// TwinCAT 3 PLC project PLC1
// ProgramVersion: 3.1.4020.4
// libraries:
//   Tc2_MC2, * (Beckhoff Automation GmbH)
//   Tc2_Standard, * (Beckhoff Automation GmbH)
//   Tc2_System, * (Beckhoff Automation GmbH)
//   Tc2_Utilities, * (Beckhoff Automation GmbH)
//   Tc3_MC2_AdvancedHoming, * (Beckhoff Automation GmbH)
//   Tc3_Module, * (Beckhoff Automation GmbH)
//   Festo TcMC Library for TwinCAT 3,3.1.1,Festo AG & Co. KG
// project tree:
//   DataType/ MoveState_t.TcDUT
//   / PlcTask.TcTTO (not stored)
//   POUs/ AxisCtrl.TcPOU, MAIN.TcPOU
// real-time tasks:
//   TASK PlcTask: cycle T#10ms, priority 20, ADS port 350
// motion (NC):
//   TASK NC-Task 1 SAF: cycle T#2ms, priority 4, ADS port 501
//   TASK NC-Task 1 SVB: cycle T#10ms, priority 8, ADS port 511
//   AXIS Axis 1 (id 1)
//     Dynamic: AccelerationMaximum=20000, DecelerationMaximum=20000, Acceleration=10000, Deceleration=10000, Jerk=200000
//     Velo: FastManual=300, Maximum=1000
//     OtherSettings: AllowMotionCmdToSlave=true
//     encoder EncType=19
//       EncPara: ScaleFactorNumerator=90, ScaleFactorDenominator=65536, MaxCount=#xffffffff
//         Inc: RefSearchInverse=true, RefMode=5
//     drive DrvType=16
//       DrvPara: MaxCount=#xffffffff, DriveControlDWord=#x00000100
//         Analog: VeloReferenz=1100
//         TimeComp: TaskDelayCycles=1
//     controller CtrType=1
//       CtrPara: PriorControlFactor=1
//         Observer: BandWidth=20
//   AXIS Axis 2 (id 2)
//     Dynamic: AccelerationMaximum=20000, DecelerationMaximum=20000, Acceleration=10000, Deceleration=10000, Jerk=200000
//     Velo: Maximum=1000
//     OtherSettings: AllowMotionCmdToSlave=true
//     encoder EncType=19
//       EncPara: ScaleFactorNumerator=90, ScaleFactorDenominator=65536, MaxCount=#xffffffff
//         Inc: RefSearchInverse=true
//     drive DrvType=16
//       DrvPara: MaxCount=#xffffffff, DriveControlDWord=#x00000100
//         Analog: VeloReferenz=1100
//         TimeComp: TaskDelayCycles=1
//     controller CtrType=1
//       CtrPara: PriorControlFactor=1
//         Observer: BandWidth=20
//   AXIS Axis 3 (id 3)
//     Dynamic: AccelerationMaximum=20000, DecelerationMaximum=20000, Acceleration=10000, Deceleration=10000, Jerk=200000
//     Velo: Maximum=1000
//     OtherSettings: AllowMotionCmdToSlave=true
//     encoder EncType=1
//       EncPara: ScaleFactorNumerator=90, ScaleFactorDenominator=65536
//         Inc: RefSearchInverse=true
//     drive DrvType=5
//       Analog: VeloReferenz=1100
//       TimeComp: TaskDelayCycles=1
//     controller CtrType=1
//       CtrPara: PriorControlFactor=1
//         Observer: BandWidth=20
//   AXIS Axis 4 (id 4)
//     Dynamic: AccelerationMaximum=20000, DecelerationMaximum=20000, Acceleration=10000, Deceleration=10000, Jerk=200000
//     Velo: Maximum=1000
//     OtherSettings: AllowMotionCmdToSlave=true
//     encoder EncType=1
//       EncPara: ScaleFactorNumerator=90, ScaleFactorDenominator=65536
//         Inc: RefSearchInverse=true
//     drive DrvType=5
//       Analog: VeloReferenz=1100
//       TimeComp: TaskDelayCycles=1
//     controller CtrType=1
//       CtrPara: PriorControlFactor=1
//         Observer: BandWidth=20
//   AXIS Axis 5 (id 5)
//     Dynamic: AccelerationMaximum=20000, DecelerationMaximum=20000, Acceleration=10000, Deceleration=10000, Jerk=200000
//     Velo: Maximum=1000
//     OtherSettings: AllowMotionCmdToSlave=true
//     encoder EncType=1
//       EncPara: ScaleFactorNumerator=90, ScaleFactorDenominator=65536
//         Inc: RefSearchInverse=true
//     drive DrvType=5
//       Analog: VeloReferenz=1100
//       TimeComp: TaskDelayCycles=1
//     controller CtrType=1
//       CtrPara: PriorControlFactor=1
//         Observer: BandWidth=20
//   AXIS Axis 6 (id 6)
//     Dynamic: AccelerationMaximum=20000, DecelerationMaximum=20000, Acceleration=10000, Deceleration=10000, Jerk=200000
//     Velo: Maximum=1000
//     OtherSettings: AllowMotionCmdToSlave=true
//     encoder EncType=1
//       EncPara: ScaleFactorNumerator=90, ScaleFactorDenominator=65536
//         Inc: RefSearchInverse=true
//     drive DrvType=5
//       Analog: VeloReferenz=1100
//       TimeComp: TaskDelayCycles=1
//     controller CtrType=1
//       CtrPara: PriorControlFactor=1
//         Observer: BandWidth=20
//   AXIS Axis 7 (id 7)
//     Dynamic: AccelerationMaximum=20000, DecelerationMaximum=20000, Acceleration=10000, Deceleration=10000, Jerk=200000
//     Velo: Maximum=1000
//     OtherSettings: AllowMotionCmdToSlave=true
//     encoder EncType=1
//       EncPara: ScaleFactorNumerator=90, ScaleFactorDenominator=65536
//         Inc: RefSearchInverse=true
//     drive DrvType=5
//       Analog: VeloReferenz=1100
//       TimeComp: TaskDelayCycles=1
//     controller CtrType=1
//       CtrPara: PriorControlFactor=1
//         Observer: BandWidth=20
//   AXIS Axis 8 (id 8)
//     Dynamic: AccelerationMaximum=20000, DecelerationMaximum=20000, Acceleration=10000, Deceleration=10000, Jerk=200000
//     Velo: Maximum=1000
//     OtherSettings: AllowMotionCmdToSlave=true
//     encoder EncType=1
//       EncPara: ScaleFactorNumerator=90, ScaleFactorDenominator=65536
//         Inc: RefSearchInverse=true
//     drive DrvType=5
//       Analog: VeloReferenz=1100
//       TimeComp: TaskDelayCycles=1
//     controller CtrType=1
//       CtrPara: PriorControlFactor=1
//         Observer: BandWidth=20
//   AXIS Axis 9 (id 9)
//     Dynamic: AccelerationMaximum=20000, DecelerationMaximum=20000, Acceleration=10000, Deceleration=10000, Jerk=200000
//     Velo: Maximum=1000
//     OtherSettings: AllowMotionCmdToSlave=true
//     encoder EncType=1
//       EncPara: ScaleFactorNumerator=90, ScaleFactorDenominator=65536
//         Inc: RefSearchInverse=true
//     drive DrvType=5
//       Analog: VeloReferenz=1100
//       TimeComp: TaskDelayCycles=1
//     controller CtrType=1
//       CtrPara: PriorControlFactor=1
//         Observer: BandWidth=20
//   AXIS Axis 10 (id 10)
//     Dynamic: AccelerationMaximum=20000, DecelerationMaximum=20000, Acceleration=10000, Deceleration=10000, Jerk=200000
//     Velo: Maximum=1000
//     OtherSettings: AllowMotionCmdToSlave=true
//     encoder EncType=1
//       EncPara: ScaleFactorNumerator=90, ScaleFactorDenominator=65536
//         Inc: RefSearchInverse=true
//     drive DrvType=5
//       Analog: VeloReferenz=1100
//       TimeComp: TaskDelayCycles=1
//     controller CtrType=1
//       CtrPara: PriorControlFactor=1
//         Observer: BandWidth=20
// I/O:
//   DEVICE NIC, AmsNetId 192.168.2.43.2.1
//     Ctr1 [CMMP-AS V4p0 CiA402]
//     Ctr2 [CMMP-AS V4p0 CiA402]
// variable links:
//   NC-Task 1 SAF/Axes/Axis 1 <-> NIC/Ctr1
//     Drive/Inputs/In/nDataIn1 <-> Inputs_1/Following_Error_Actual_Value
//     Drive/Inputs/In/nDcOutputTime <-> InfoData/DcOutputShift
//     Drive/Inputs/In/nState1 <-> Inputs/Statusword
//     Drive/Inputs/In/nState2 <-> Inputs/Statusword @bit 8
//     Drive/Inputs/In/nState4 @bit 1 <-> WcState/InputToggle
//     Drive/Inputs/In/nState4 <-> WcState/WcState
//     Drive/Outputs/Out/nCtrl1 <-> Outputs/Controlword
//     Drive/Outputs/Out/nCtrl2 <-> Outputs/Controlword @bit 8
//     Drive/Outputs/Out/nDataOut1 <-> Outputs/IP_Data_Record
//     Enc/Inputs/In/nDataIn1 <-> Inputs/Position_Actual_Value
//     Enc/Inputs/In/nDcInputTime <-> InfoData/DcInputShift
//     Enc/Inputs/In/nState4 @bit 1 <-> WcState/InputToggle
//     Enc/Inputs/In/nState4 <-> WcState/WcState
//   NC-Task 1 SAF/Axes/Axis 2 <-> NIC/Ctr2
//     Drive/Inputs/In/nDataIn1 <-> Inputs_1/Following_Error_Actual_Value
//     Drive/Inputs/In/nDcOutputTime <-> InfoData/DcOutputShift
//     Drive/Inputs/In/nState1 <-> Inputs/Statusword
//     Drive/Inputs/In/nState2 <-> Inputs/Statusword @bit 8
//     Drive/Inputs/In/nState4 @bit 1 <-> WcState/InputToggle
//     Drive/Inputs/In/nState4 <-> WcState/WcState
//     Drive/Outputs/Out/nCtrl1 <-> Outputs/Controlword
//     Drive/Outputs/Out/nCtrl2 <-> Outputs/Controlword @bit 8
//     Drive/Outputs/Out/nDataOut1 <-> Outputs/IP_Data_Record
//     Enc/Inputs/In/nDataIn1 <-> Inputs/Position_Actual_Value
//     Enc/Inputs/In/nDcInputTime <-> InfoData/DcInputShift
//     Enc/Inputs/In/nState4 @bit 1 <-> WcState/InputToggle
//     Enc/Inputs/In/nState4 <-> WcState/WcState
//   PLC1/PLC1 Instance <-> NIC/Ctr1
//     PlcTask Inputs/MAIN.axisCtrls[1].amsAddr <-> InfoData/AdsAddr
//     PlcTask Inputs/MAIN.axisCtrls[1].dig_in <-> Input3/swn
//   PLC1/PLC1 Instance <-> NIC/Ctr2
//     PlcTask Inputs/MAIN.axisCtrls[2].amsAddr <-> InfoData/AdsAddr
//   PLC1/PLC1 Instance <-> NC-Task 1 SAF/Axes/Axis 1
//     PlcTask Inputs/MAIN.axisCtrls[1].axis.NcToPlc <-> Outputs/ToPlc
//     PlcTask Outputs/MAIN.axisCtrls[1].axis.PlcToNc <-> Inputs/FromPlc
//   PLC1/PLC1 Instance <-> NC-Task 1 SAF/Axes/Axis 10
//     PlcTask Inputs/MAIN.axisCtrls[10].axis.NcToPlc <-> Outputs/ToPlc
//     PlcTask Outputs/MAIN.axisCtrls[10].axis.PlcToNc <-> Inputs/FromPlc
//   PLC1/PLC1 Instance <-> NC-Task 1 SAF/Axes/Axis 2
//     PlcTask Inputs/MAIN.axisCtrls[2].axis.NcToPlc <-> Outputs/ToPlc
//     PlcTask Outputs/MAIN.axisCtrls[2].axis.PlcToNc <-> Inputs/FromPlc
//   PLC1/PLC1 Instance <-> NC-Task 1 SAF/Axes/Axis 3
//     PlcTask Inputs/MAIN.axisCtrls[3].axis.NcToPlc <-> Outputs/ToPlc
//     PlcTask Outputs/MAIN.axisCtrls[3].axis.PlcToNc <-> Inputs/FromPlc
//   PLC1/PLC1 Instance <-> NC-Task 1 SAF/Axes/Axis 4
//     PlcTask Inputs/MAIN.axisCtrls[4].axis.NcToPlc <-> Outputs/ToPlc
//     PlcTask Outputs/MAIN.axisCtrls[4].axis.PlcToNc <-> Inputs/FromPlc
//   PLC1/PLC1 Instance <-> NC-Task 1 SAF/Axes/Axis 5
//     PlcTask Inputs/MAIN.axisCtrls[5].axis.NcToPlc <-> Outputs/ToPlc
//     PlcTask Outputs/MAIN.axisCtrls[5].axis.PlcToNc <-> Inputs/FromPlc
//   PLC1/PLC1 Instance <-> NC-Task 1 SAF/Axes/Axis 6
//     PlcTask Inputs/MAIN.axisCtrls[6].axis.NcToPlc <-> Outputs/ToPlc
//     PlcTask Outputs/MAIN.axisCtrls[6].axis.PlcToNc <-> Inputs/FromPlc
//   PLC1/PLC1 Instance <-> NC-Task 1 SAF/Axes/Axis 7
//     PlcTask Inputs/MAIN.axisCtrls[7].axis.NcToPlc <-> Outputs/ToPlc
//     PlcTask Outputs/MAIN.axisCtrls[7].axis.PlcToNc <-> Inputs/FromPlc
//   PLC1/PLC1 Instance <-> NC-Task 1 SAF/Axes/Axis 8
//     PlcTask Inputs/MAIN.axisCtrls[8].axis.NcToPlc <-> Outputs/ToPlc
//     PlcTask Outputs/MAIN.axisCtrls[8].axis.PlcToNc <-> Inputs/FromPlc
//   PLC1/PLC1 Instance <-> NC-Task 1 SAF/Axes/Axis 9
//     PlcTask Inputs/MAIN.axisCtrls[9].axis.NcToPlc <-> Outputs/ToPlc
//     PlcTask Outputs/MAIN.axisCtrls[9].axis.PlcToNc <-> Inputs/FromPlc

// ---- DataType/MoveState_t.TcDUT
TYPE MoveState_t :
(
	 MOVESTATE_RESET,
	 MOVESTATE_INIT,
	 MOVESTATE_ENABLE,
	 MOVESTATE_HOMING,
	 MOVESTATE_MOVING,
	 MOVESTATE_ERROR	
);
END_TYPE

// ---- POUs/AxisCtrl.TcPOU
FUNCTION_BLOCK AxisCtrl
VAR_INPUT
END_VAR
VAR_OUTPUT
END_VAR
VAR
	axis : AXIS_REF;
	state : MoveState_t;
	
	moveAbs: MC_MoveAbsolute;
	moveAbsOut: ST_McOutputs;

	moveAbs2: MC_MoveAbsolute;
	moveAbsOut2: ST_McOutputs;
	
	power: MC_Power;
	powerOut : ST_McOutputs;
	
	reset: MC_Reset;
	resetOut : ST_McOutputs;
	
	halt: MC_Halt;
	haltOut : ST_McOutputs;
	
	cmd_pos : LREAL;
	cmd_vel : LREAL;
	cmd_acc : LREAL;
	cmd_vel_end : LREAL;
	cmd_need_exe : BOOL;
	cmd_halt : BOOL := FALSE;
	
	readActPos: MC_ReadActualPosition;
	readActVel: MC_ReadActualVelocity;
	
	actPosOut : ST_McOutputs;
	actVelOut : ST_McOutputs;
	
	actual_pos : LREAL;
	actual_vel : LREAL;

	dig_in AT %ID0 : DINT;
	
	(*
	negative_limit_sw AT %IX0.0 : BOOL;
	positive_limit_sw AT %IX0.1 : BOOL;
	reference_sw AT %IX0.2 : BOOL;
		*)
	
	HomingExecute: BOOL := FALSE;
	HomingError : BOOL := FALSE;
	
	(* Basic Homing*)
	home: MC_Home;
	homeOut: ST_McOutputs;
	
	(* TwinCat Advanced Homing*)
	homingParameter: MC_HomingParameter;
	stepHomingParameter: MC_StepHomingParameter;
	stepHomingParameterOut : ST_McOutputs;	
	stepBlock: MC_StepBlock;
	stepBlockOut: ST_McOutputs;
	stepLimitSwitch: MC_StepLimitSwitch;
	stepLimitSwitchOut: ST_McOutputs;
	finishHoming: MC_FinishHoming;
	finishHomingOut : ST_McOutputs;
	
	homeOption2: ST_Home_Options2;
	homeOption3: ST_Home_Options3;
	
	(* Festo Homing*)
	homeFesto: Festo_MC_Home;
	homeFestoOut : ST_McOutputs;
	
	amsAddr AT %I* : AMSADDR;
	deviceNetID	:T_AmsNetId	:= '192.168.2.43.2.1';
	
	
	driveError: Festo_GetDriveError;
	// variables for function block "Festo_GetDriveError"
	GetErrorEnable		:BOOL;
	GetErrorBusy		:BOOL;
	DriveInErrorState	:BOOL;
	DriveErrorNumber	:ARRAY [1..4] OF DWORD;
	GetErrorWasAbortive	:BOOL;
	GetErrorId	: UDINT;

END_VAR

	axis.ReadStatus();
	
	CASE state OF
		
		MOVESTATE_INIT :
			moveAbs.Execute := FALSE;
			reset.Execute := FALSE;
			power.Enable := FALSE;
			
			state := MOVESTATE_ENABLE;
		MOVESTATE_ENABLE:
			power.Enable := TRUE;
			
			IF power.Status THEN
				state := MOVESTATE_HOMING;
			ELSIF power.Error THEN
				state := MOVESTATE_ERROR;
			END_IF
			
		MOVESTATE_HOMING:

			IF axis.Status.Homed THEN
			 	HomingExecute := FALSE;
				state := MOVESTATE_MOVING;				
			ELSE
				HomingExecute := TRUE;				
			END_IF
		
		MOVESTATE_MOVING:		
			IF cmd_need_exe THEN
				IF moveAbs.Busy THEN
					moveAbs2.Position := cmd_pos;
					moveAbs2.Velocity := cmd_vel;
					moveAbs2.BufferMode := MC_Aborting;
					moveAbs2.Execute := TRUE;
				ELSE
					moveAbs.Position := cmd_pos;
					moveAbs.Velocity := cmd_vel;
					moveAbs.BufferMode := MC_Aborting;
					moveAbs.Execute := TRUE;
				END_IF;		
				
				cmd_need_exe := FALSE;
			END_IF;		
		
			IF moveAbs.Done THEN
				moveAbs.Execute := FALSE;
			ELSIF moveAbs.CommandAborted THEN
				moveAbs.Execute := FALSE;
			ELSIF moveAbs.Error THEN
				state := MOVESTATE_ERROR;
			END_IF
			
			
			IF moveAbs2.Done THEN
				moveAbs2.Execute := FALSE;
			ELSIF moveAbs2.CommandAborted THEN
				moveAbs2.Execute := FALSE;
			ELSIF moveAbs2.Error THEN
				state := MOVESTATE_ERROR;
			END_IF
			
		MOVESTATE_ERROR :
			IF axis.Status.Error THEN
				state := MOVESTATE_RESET;
			ELSE
				state := MOVESTATE_INIT;
			END_IF

		MOVESTATE_RESET :
			reset.Execute := TRUE;
			IF reset.Done THEN
				state := MOVESTATE_INIT;
			ELSIF reset.Error THEN
				state := MOVESTATE_INIT;
			END_IF
	END_CASE
	
	
	ActPower();
	ActMove();
	ActReset();
	ActRead();
	ActHalt();
	(*ActHome();*)
	(*ActHomeBlock(); *)
	(*ActHomeLimit(); *)
	ActHomeFesto();
	
	IF haltOut.Done OR haltOut.Error THEN
		cmd_halt := FALSE;
	END_IF

ACTION ActHalt:
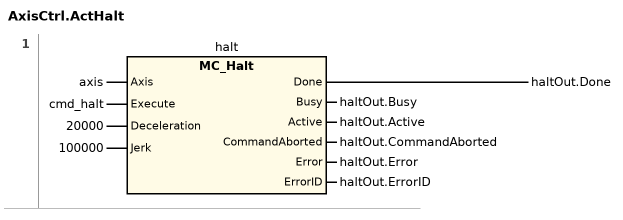
// NETWORK 1
halt(
    Axis := axis,
    Execute := cmd_halt,
    Deceleration := 20000,
    Jerk := 100000,
    Busy => haltOut.Busy,
    Active => haltOut.Active,
    CommandAborted => haltOut.CommandAborted,
    Error => haltOut.Error,
    ErrorID => haltOut.ErrorID); // MC_Halt
haltOut.Done := halt.Done;
END_ACTION

ACTION ActHome:
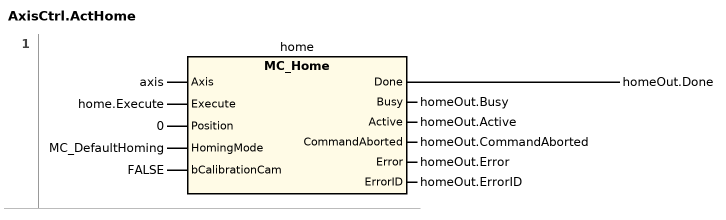
// NETWORK 1
home(
    Axis := axis,
    Execute := home.Execute,
    Position := 0,
    HomingMode := MC_DefaultHoming,
    bCalibrationCam := FALSE,
    Busy => homeOut.Busy,
    Active => homeOut.Active,
    CommandAborted => homeOut.CommandAborted,
    Error => homeOut.Error,
    ErrorID => homeOut.ErrorID); // MC_Home
homeOut.Done := home.Done;
END_ACTION

ACTION ActHomeBlock:
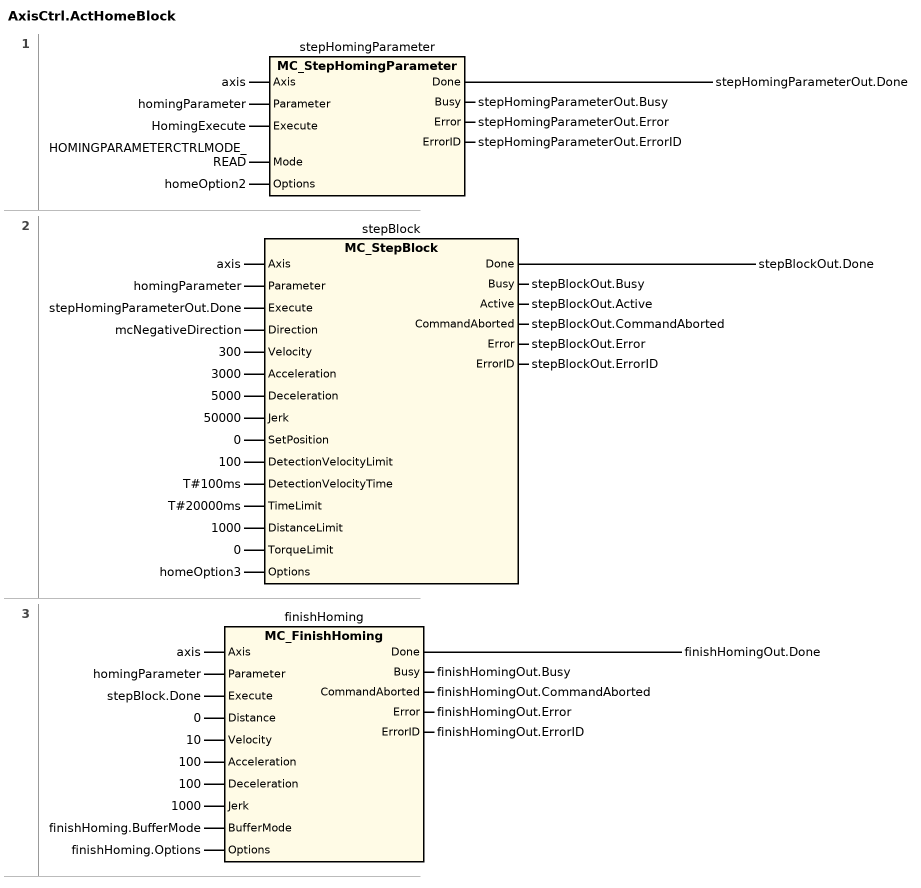
// NETWORK 1
stepHomingParameter(
    Axis := axis,
    Parameter := homingParameter,
    Execute := HomingExecute,
    Mode := HOMINGPARAMETERCTRLMODE_READ,
    Options := homeOption2,
    Busy => stepHomingParameterOut.Busy,
    Error => stepHomingParameterOut.Error,
    ErrorID => stepHomingParameterOut.ErrorID); // MC_StepHomingParameter
stepHomingParameterOut.Done := stepHomingParameter.Done;

// NETWORK 2
stepBlock(
    Axis := axis,
    Parameter := homingParameter,
    Execute := stepHomingParameterOut.Done,
    Direction := mcNegativeDirection,
    Velocity := 300,
    Acceleration := 3000,
    Deceleration := 5000,
    Jerk := 50000,
    SetPosition := 0,
    DetectionVelocityLimit := 100,
    DetectionVelocityTime := T#100ms,
    TimeLimit := T#20000ms,
    DistanceLimit := 1000,
    TorqueLimit := 0,
    Options := homeOption3,
    Busy => stepBlockOut.Busy,
    Active => stepBlockOut.Active,
    CommandAborted => stepBlockOut.CommandAborted,
    Error => stepBlockOut.Error,
    ErrorID => stepBlockOut.ErrorID); // MC_StepBlock
stepBlockOut.Done := stepBlock.Done;

// NETWORK 3
finishHoming(
    Axis := axis,
    Parameter := homingParameter,
    Execute := stepBlock.Done,
    Distance := 0,
    Velocity := 10,
    Acceleration := 100,
    Deceleration := 100,
    Jerk := 1000,
    BufferMode := finishHoming.BufferMode,
    Options := finishHoming.Options,
    Busy => finishHomingOut.Busy,
    CommandAborted => finishHomingOut.CommandAborted,
    Error => finishHomingOut.Error,
    ErrorID => finishHomingOut.ErrorID); // MC_FinishHoming
finishHomingOut.Done := finishHoming.Done;
END_ACTION

ACTION ActHomeFesto:
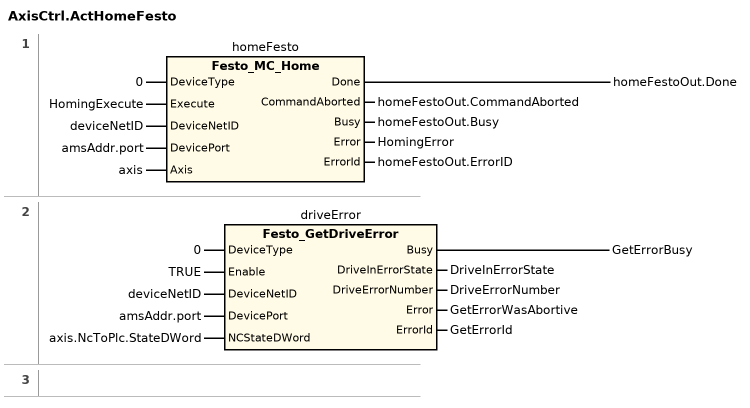
// NETWORK 1
homeFesto(
    DeviceType := 0,
    Execute := HomingExecute,
    DeviceNetID := deviceNetID,
    DevicePort := amsAddr.port,
    Axis := axis,
    CommandAborted => homeFestoOut.CommandAborted,
    Busy => homeFestoOut.Busy,
    Error => HomingError,
    ErrorId => homeFestoOut.ErrorID); // Festo_MC_Home
homeFestoOut.Done := homeFesto.Done;

// NETWORK 2
driveError(
    DeviceType := 0,
    Enable := TRUE,
    DeviceNetID := deviceNetID,
    DevicePort := amsAddr.port,
    NCStateDWord := axis.NcToPlc.StateDWord,
    DriveInErrorState => DriveInErrorState,
    DriveErrorNumber => DriveErrorNumber,
    Error => GetErrorWasAbortive,
    ErrorId => GetErrorId); // Festo_GetDriveError
GetErrorBusy := driveError.Busy;

// NETWORK 3
END_ACTION

ACTION ActHomeLimit:
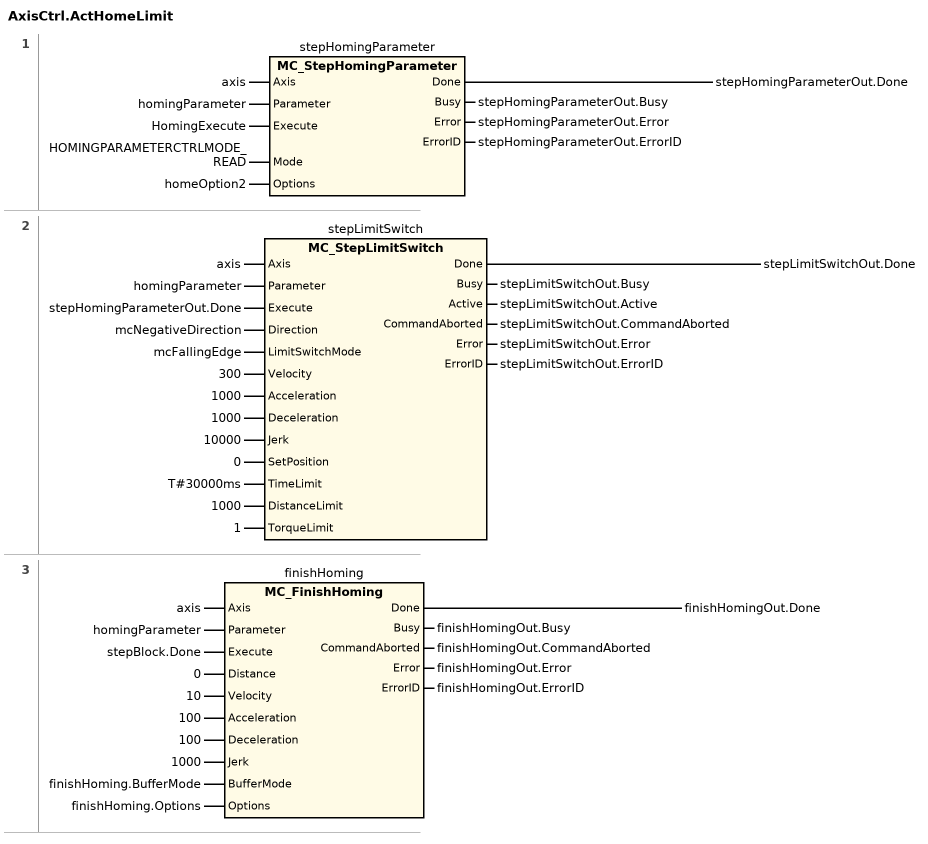
// NETWORK 1
stepHomingParameter(
    Axis := axis,
    Parameter := homingParameter,
    Execute := HomingExecute,
    Mode := HOMINGPARAMETERCTRLMODE_READ,
    Options := homeOption2,
    Busy => stepHomingParameterOut.Busy,
    Error => stepHomingParameterOut.Error,
    ErrorID => stepHomingParameterOut.ErrorID); // MC_StepHomingParameter
stepHomingParameterOut.Done := stepHomingParameter.Done;

// NETWORK 2
stepLimitSwitch(
    Axis := axis,
    Parameter := homingParameter,
    Execute := stepHomingParameterOut.Done,
    Direction := mcNegativeDirection,
    LimitSwitchMode := mcFallingEdge,
    Velocity := 300,
    Acceleration := 1000,
    Deceleration := 1000,
    Jerk := 10000,
    SetPosition := 0,
    TimeLimit := T#30000ms,
    DistanceLimit := 1000,
    TorqueLimit := 1,
    Busy => stepLimitSwitchOut.Busy,
    Active => stepLimitSwitchOut.Active,
    CommandAborted => stepLimitSwitchOut.CommandAborted,
    Error => stepLimitSwitchOut.Error,
    ErrorID => stepLimitSwitchOut.ErrorID); // MC_StepLimitSwitch
stepLimitSwitchOut.Done := stepLimitSwitch.Done;

// NETWORK 3
finishHoming(
    Axis := axis,
    Parameter := homingParameter,
    Execute := stepBlock.Done,
    Distance := 0,
    Velocity := 10,
    Acceleration := 100,
    Deceleration := 100,
    Jerk := 1000,
    BufferMode := finishHoming.BufferMode,
    Options := finishHoming.Options,
    Busy => finishHomingOut.Busy,
    CommandAborted => finishHomingOut.CommandAborted,
    Error => finishHomingOut.Error,
    ErrorID => finishHomingOut.ErrorID); // MC_FinishHoming
finishHomingOut.Done := finishHoming.Done;
END_ACTION

ACTION ActMove:
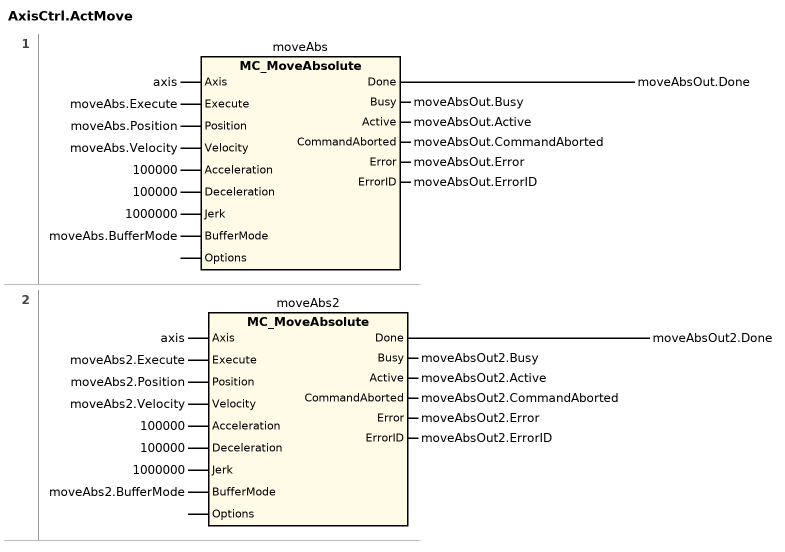
// NETWORK 1
moveAbs(
    Axis := axis,
    Execute := moveAbs.Execute,
    Position := moveAbs.Position,
    Velocity := moveAbs.Velocity,
    Acceleration := 100000,
    Deceleration := 100000,
    Jerk := 1000000,
    BufferMode := moveAbs.BufferMode,
    Busy => moveAbsOut.Busy,
    Active => moveAbsOut.Active,
    CommandAborted => moveAbsOut.CommandAborted,
    Error => moveAbsOut.Error,
    ErrorID => moveAbsOut.ErrorID); // MC_MoveAbsolute
moveAbsOut.Done := moveAbs.Done;

// NETWORK 2
moveAbs2(
    Axis := axis,
    Execute := moveAbs2.Execute,
    Position := moveAbs2.Position,
    Velocity := moveAbs2.Velocity,
    Acceleration := 100000,
    Deceleration := 100000,
    Jerk := 1000000,
    BufferMode := moveAbs2.BufferMode,
    Busy => moveAbsOut2.Busy,
    Active => moveAbsOut2.Active,
    CommandAborted => moveAbsOut2.CommandAborted,
    Error => moveAbsOut2.Error,
    ErrorID => moveAbsOut2.ErrorID); // MC_MoveAbsolute
moveAbsOut2.Done := moveAbs2.Done;
END_ACTION

ACTION ActPower:
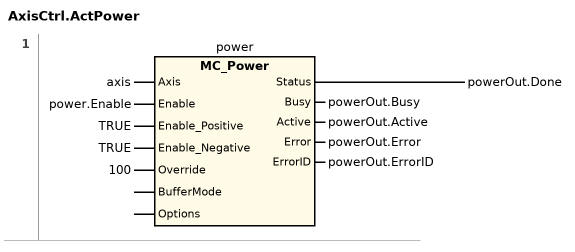
// NETWORK 1
power(
    Axis := axis,
    Enable := power.Enable,
    Enable_Positive := TRUE,
    Enable_Negative := TRUE,
    Override := 100,
    Busy => powerOut.Busy,
    Active => powerOut.Active,
    Error => powerOut.Error,
    ErrorID => powerOut.ErrorID); // MC_Power
powerOut.Done := power.Status;
END_ACTION

ACTION ActRead:
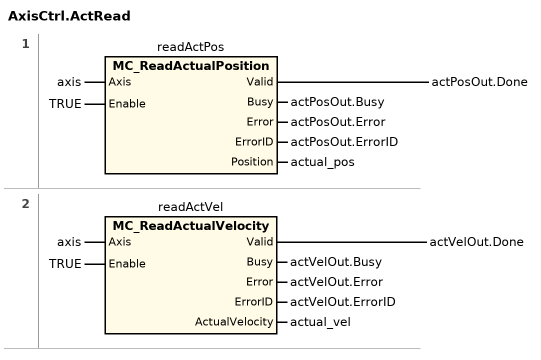
// NETWORK 1
readActPos(
    Axis := axis,
    Enable := TRUE,
    Busy => actPosOut.Busy,
    Error => actPosOut.Error,
    ErrorID => actPosOut.ErrorID,
    Position => actual_pos); // MC_ReadActualPosition
actPosOut.Done := readActPos.Valid;

// NETWORK 2
readActVel(
    Axis := axis,
    Enable := TRUE,
    Busy => actVelOut.Busy,
    Error => actVelOut.Error,
    ErrorID => actVelOut.ErrorID,
    ActualVelocity => actual_vel); // MC_ReadActualVelocity
actVelOut.Done := readActVel.Valid;
END_ACTION

ACTION ActReset:
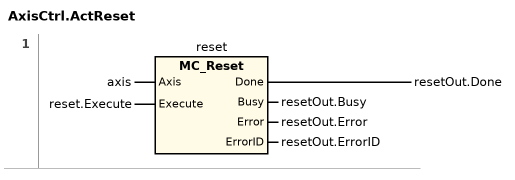
// NETWORK 1
reset(
    Axis := axis,
    Execute := reset.Execute,
    Busy => resetOut.Busy,
    Error => resetOut.Error,
    ErrorID => resetOut.ErrorID); // MC_Reset
resetOut.Done := reset.Done;
END_ACTION

END_FUNCTION_BLOCK

// ---- POUs/MAIN.TcPOU
PROGRAM MAIN
VAR
	axisCtrls : ARRAY[1 .. 10] OF AxisCtrl;
	i : INT := 0;
END_VAR

FOR i := 1 TO 10 DO
 	axisCtrls[i]();
END_FOR;

END_PROGRAM
